SUBAPPLICATION Uebung_010a5_AX (* SoftKey_F1 auf DigitalOutput_Q1 (Datapanel) *)
  (* Standard: 61499-2; Description: Copyright (c) 2023 Meisterschulen am Ostbahnhof This program and the accompanying materials are made available under the terms of the Eclipse Public License 2.0 which is available at https://www.eclipse.org/legal/epl-2.0/ SPDX-License-Identifier: EPL-2.0 *)
  (* Version 1.0, 2023-10-23, Franz Höpfinger, Meisterschulen am Ostbahnhof, initial API and implementation and/or initial documentation *)
  PACKAGE Uebungen;
  IMPORT DataPanel::io::MI::DQ::DataPanel_MI_DO::Input_Power_Port_5;
  IMPORT DataPanel::io::MI::const::MI::MI_00;
  IMPORT Uebungen::const::UT::DefaultPool::SoftKey_F1;
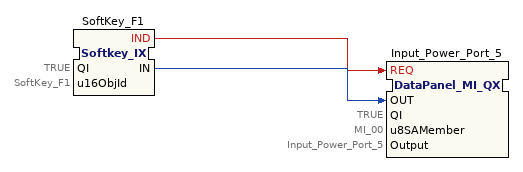
  FBS
    Input_Power_Port_5 : DataPanel::io::MI::DQ::DataPanel_MI_QX(QI := TRUE, u8SAMember := MI_00, Output := Input_Power_Port_5);
    SoftKey_F1 : isobus::UT::io::Softkey::Softkey_IX(QI := TRUE, u16ObjId := SoftKey_F1);
  END_FBS
  EVENT_CONNECTIONS
    SoftKey_F1.IND TO Input_Power_Port_5.REQ;
  END_CONNECTIONS
  DATA_CONNECTIONS
    SoftKey_F1.IN TO Input_Power_Port_5.OUT;
  END_CONNECTIONS
END_SUBAPPLICATION
